// TIA Portal V16 export
// export: Created 2021-08-23T11:40:58.8156124Z, ExportSetting WithDefaults, DisplayName Totally Integrated Automation Portal, DisplayVersion V16 Update 4, DisplayName TIA Portal Version Control Interface, DisplayVersion V16 Update 2, DisplayName TIA Portal Openness, DisplayVersion V16 Update 4, DisplayName STEP 7 Professional, DisplayVersion V16 Update 4, DisplayName STEP 7 Safety, DisplayVersion V16, DisplayName WinCC Advanced, DisplayVersion V16 Update 4
ORGANIZATION_BLOCK "Main"   // OB1, LAD, ProgramCycle
TITLE = "Main Program Sweep (Cycle)"
{ S7_Optimized_Access := 'TRUE' }
VERSION : 0.1
// stored: AutoNumber true, IsIECCheckEnabled false, SetENOAutomatically false
   VAR_INPUT
      Initial_Call : Bool;   // Initial call of this OB
      Remanence : Bool;   // =True, if remanent data are available
   END_VAR
   VAR_TEMP
      tTemp1 : Bool;
      tTemp2 : Bool;
   END_VAR
BEGIN

REGION Network 1: Komentarz
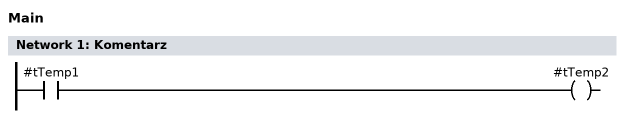
   RUNG wire#powerrail
      Contact( #tTemp1 )
      Coil( #tTemp2 )
   END_RUNG
   // the same network as SCL:
   #tTemp2 := #tTemp1;
END_REGION
END_ORGANIZATION_BLOCK
